// TIA Portal project "babu_timer3lamps" (V15)

(* hardware
DEVICE "S7-1200 station_1"  S7-1200 Station
   slot 0: "Rack_0"  S7-1200 Rack  Rack  V1.0
   slot 1: "PLC_1"  CPU 1212C DC/DC/DC  6ES7 212-1AE40-0XB0  V4.2
*)

// ===== PLC "PLC_1"  CPU 1212C DC/DC/DC =====

VAR_GLOBAL   // PLC tag table "Tag table_1"
   "SWITCH 1" AT %M0.0 : Bool;
   "LAMP 1" AT %Q0.1 : Bool;
   "LAMP 2" AT %Q0.2 : Bool;
   "LAMP 3" AT %Q0.3 : Bool;
   "MEMORY 1" AT %M0.4 : Bool;
   "MEMORY 2" AT %M0.5 : Bool;
END_VAR

// folder: System blocks/Program resources

DATA_BLOCK "IEC_Timer_0_DB"   // DB1
{ S7_Optimized_Access := 'TRUE' }
AUTHOR : Simatic
FAMILY : IEC
NAME : IEC_TMR
VERSION : 1.0
// stored: InstanceOfName IEC_TIMER
"IEC_TIMER"
BEGIN
END_DATA_BLOCK

DATA_BLOCK "IEC_Timer_0_DB_1"   // DB2
{ S7_Optimized_Access := 'TRUE' }
AUTHOR : Simatic
FAMILY : IEC
NAME : IEC_TMR
VERSION : 1.0
// stored: InstanceOfName IEC_TIMER
"IEC_TIMER"
BEGIN
END_DATA_BLOCK

// folder: (top level)

ORGANIZATION_BLOCK "Main"   // OB1, LAD, ProgramCycle
TITLE = "Main Program Sweep (Cycle)"
{ S7_Optimized_Access := 'TRUE' }
VERSION : 0.1
   VAR_INPUT
      Initial_Call : Bool;   // Initial call of this OB
      Remanence : Bool;   // =True, if remanent data are available
   END_VAR
BEGIN

REGION Network 1
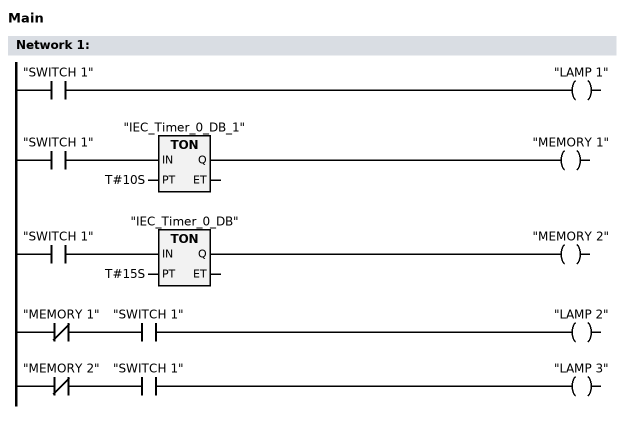
   "LAMP 1" := "SWITCH 1";
   "IEC_Timer_0_DB_1".TON(IN := "SWITCH 1", PT := T#10S);
   "MEMORY 1" := "IEC_Timer_0_DB_1".Q;
   "IEC_Timer_0_DB".TON(IN := "SWITCH 1", PT := T#15S);
   "MEMORY 2" := "IEC_Timer_0_DB".Q;
   "LAMP 2" := NOT "MEMORY 1" AND "SWITCH 1";
   "LAMP 3" := NOT "MEMORY 2" AND "SWITCH 1";
END_REGION
END_ORGANIZATION_BLOCK